PROGRAM POU_Process_Deneme
VAR
	nStateProcess: INT;
	bSystemStart: BOOL;
	bSensor: BOOL;
	T1: TON;
	T2: TON;
	rtrig_Obj: R_TRIG;
END_VAR

		
	stAxisM1_B.In.xEnable	:= TRUE;
	stAxisM2_C.In.xEnable	:= TRUE;
	stAxisM3_A.In.xEnable	:= TRUE;
	
	stAxisX.In.xEnable	:= TRUE;
	stAxisY.In.xEnable	:= TRUE;
	stAxisZ.In.xEnable	:= TRUE;
		
	stAxisM1_B.In.fOverride	:= 100;
	stAxisM2_C.In.fOverride	:= 100;
	stAxisM3_A.In.fOverride	:= 100;
	
	stAxisX.In.fOverride	:= 100;
	stAxisY.In.fOverride	:= 100;
	stAxisZ.In.fOverride	:= 100;
	

	
CASE nStateProcess	OF
	
0:
IF bSystemStart THEN


	PRG_Kinematic.bExecuteKinConfigGroup	:=	TRUE;
	stAxisX.In.xMove	:=	TRUE;
	stAxisY.In.xMove	:=	TRUE;
	stAxisZ.In.xMove	:=	TRUE;

			
	stAxisX.In.fSetVelo	:=50;
	stAxisY.In.fSetVelo	:=50;
	stAxisZ.In.fSetVelo	:=50;

	IF 
	PRG_Kinematic.fbKinConfigGroup.bDone AND 
	stAxisX.Out.xEnabled	AND
	stAxisY.Out.xEnabled	AND
	stAxisZ.Out.xEnabled	THEN
	
	

		nStateProcess	:=	10;
	
	ELSIF	PRG_Kinematic.fbKinConfigGroup.bError THEN
		nStateProcess	:=	1000;
	END_IF	
	
END_IF

10:
GVL_Process_Deneme.bMovementDone	:=	FALSE;
GVL_Process_Deneme.bDataComp	:=FALSE;


IF	GVL_Process_Deneme.bSensor	THEN
	
	GVL_Process_Deneme.bMovementDone	:=	TRUE;
	
	stAxisX.In.fSetPos	:=	0;
	stAxisY.In.fSetPos	:=	0;
	stAxisZ.In.fSetPos	:=	-400;
	

	IF 	stAxisX.Out.xMoveDone	AND stAxisY.Out.xMoveDone	AND stAxisZ.Out.xMoveDone THEN 
	
	GVL_Process_Deneme.bCatch	:=	TRUE;
	
	GVL_Process_Deneme.bMovementDone	:=	FALSE;				//Malzeme Alındı


	
	nStateProcess	:=	20;
	
	ELSIF stAxisX.Out.xAxisError	OR
	stAxisY.Out.xAxisError	OR
	stAxisZ.Out.xAxisError	OR
	stAxisM1_B.Out.xAxisError	OR
	stAxisM2_C.Out.xAxisError	OR	
	stAxisM3_A.Out.xAxisError	THEN

	nStateProcess	:=	999;	
	
END_IF
	
	
	
END_IF

20:

stAxisX.In.fSetVelo	:=300;
stAxisY.In.fSetVelo	:=300;
stAxisZ.In.fSetVelo	:=300;


stAxisZ.In.fSetPos	:=	-370;			//Alınan malzeme bırakılacağı konuma götürüldü
stAxisY.In.fSetPos	:=	310;

nStateProcess	:=	25;


25:

	IF  stAxisY.Out.xMoveDone	AND stAxisZ.Out.xMoveDone THEN 

	
	nStateProcess	:=	30;
	
	ELSIF stAxisX.Out.xAxisError	OR
	stAxisY.Out.xAxisError	OR
	stAxisZ.Out.xAxisError	OR
	stAxisM1_B.Out.xAxisError	OR
	stAxisM2_C.Out.xAxisError	OR	
	stAxisM3_A.Out.xAxisError	THEN

	nStateProcess	:=	999;	
	
END_IF
	
30:
stAxisX.In.fSetVelo	:=50;
stAxisY.In.fSetVelo	:=50;
stAxisZ.In.fSetVelo	:=50;

stAxisZ.In.fSetPos	:=	-400;		



	IF stAxisZ.Out.xMoveDone THEN 

	GVL_Process_Deneme.bDataComp	:=	TRUE;	// Malzeme bırakıldı
	
//	GVL_Process_Deneme.bMovementDone	:=	TRUE;

	GVL_Process_Deneme.bCatch	:=	FALSE;
	
	
	nStateProcess	:=	40;
	
	
	ELSIF stAxisX.Out.xAxisError	OR
	stAxisY.Out.xAxisError	OR
	stAxisZ.Out.xAxisError	OR
	stAxisM1_B.Out.xAxisError	OR
	stAxisM2_C.Out.xAxisError	OR	
	stAxisM3_A.Out.xAxisError	THEN

	nStateProcess	:=	999;	
	
END_IF


40:

stAxisX.In.fSetVelo	:=1000;
stAxisY.In.fSetVelo	:=1000;
stAxisZ.In.fSetVelo	:=1000;


stAxisX.In.fSetPos	:=	0;
stAxisY.In.fSetPos	:=	0;
stAxisZ.In.fSetPos	:=	-370;

nStateProcess	:=	45;

45:
		
	IF 	stAxisX.Out.xMoveDone	AND stAxisY.Out.xMoveDone	 THEN 


	GVL_Process_Deneme.bDataComp	:=FALSE;
		GVL_Process_Deneme.bMovementDone	:=FALSE;

	
	nStateProcess	:=	0;
	
	
	ELSIF stAxisX.Out.xAxisError	OR
	stAxisY.Out.xAxisError	OR
	stAxisZ.Out.xAxisError	OR
	stAxisM1_B.Out.xAxisError	OR
	stAxisM2_C.Out.xAxisError	OR	
	stAxisM3_A.Out.xAxisError	THEN

	nStateProcess	:=	999;	
	
END_IF





END_CASE

END_PROGRAM

(* stored: Version 1.1.0.1, ProductVersion 3.1.4024.0
   POU POU_Process_Deneme: Id {96d46232-4b1f-462f-b400-9fcb212730d7}, SpecialFunc None *)
